ABB RAPID module: 000679EB

MODULE Module1
    CONST robtarget pBaseOrigen:=[[1500,-500,750],[0,0,1,0],[0,0,0,0],[9E+09,9E+09,9E+09,9E+09,9E+09,9E+09]];
    CONST robtarget pCentroDestino:=[[1700,1000,750],[0,0,1,0],[0,0,0,0],[9E+09,9E+09,9E+09,9E+09,9E+09,9E+09]];
    CONST robtarget pReposo:=[[1808.910161514,0,1855],[0.5,0,0.866025404,0],[0,0,0,0],[9E+09,9E+09,9E+09,9E+09,9E+09,9E+09]];

ENDMODULE
